{attribute 'qualified_only'}
{attribute 'strict'}
{attribute 'to_string'}
TYPE eTransitions :
(
	Configure := 0,
	Activate:=1,
	Deactivate:=2,
	Cleanup:=3,
	Shutdown:=4,
	Destroy:=5
);
END_TYPE

(* stored: Version 1.1.0.1, ProductVersion 3.1.4026.18
   DUT eTransitions: Id {e4152442-29eb-48a3-b1e9-66669e77581f} *)
